TYPE ST_Kistler_Status :
STRUCT
    bReady       	: BOOL;
    bBusy        	: BOOL;
    bDone        	: BOOL;
    bError       	: BOOL;
    bInPosition  	: BOOL;

    bPartOK      	: BOOL;
    bPartNOK     	: BOOL;
	
	rLiveDistance 	: REAL;
	rLiveForce      : REAL;

    eKistlerState 	: E_KistlerState;
	
	// Configured evaluation limits
	rDistanceMin 	: REAL;
	rDistanceMax 	: REAL;
	rForceMin    	: REAL;
	rForceMax    	: REAL;
	
	END_STRUCT
END_TYPE

(* stored: Version 1.1.0.1
   DUT ST_Kistler_Status: Id {13fe1f7e-c843-4ff0-b94a-cef6c7ea4e07} *)
